{attribute addProperty BoxType "AX8206-0100-0101-0101"}
{attribute addProperty Id "DeviceDevice_F82A60211620Device_SafetyDevice_Safety_AF71BE9D160200Ch_ACh_A_359CD49A176220Ch_BCh_B_71B491C3176220WcStateAT %I*WcState_DC9C971540.50InfoDataAT %I*InfoData_17277C5A208260"}
{attribute addProperty CRC "932077249"}
{attribute addProperty SizeInBites "740"}
{attribute addProperty SizeInBytes "92.5"}
TYPE AX8206_36A80AF0 :
STRUCT
	{attribute addProperty Name "Device"}
	Device : Device_F82A6021;
	{attribute addProperty Name "Device_Safety"}
	Device_Safety : Device_Safety_AF71BE9D;
	{attribute addProperty Name "Ch_A"}
	Ch_A : Ch_A_359CD49A;
	{attribute addProperty Name "Ch_B"}
	Ch_B : Ch_B_71B491C3;
	{attribute addProperty Name "WcState"}
	WcState : WcState_DC9C9715;
	{attribute addProperty Name "InfoData"}
	InfoData : InfoData_17277C5A;
END_STRUCT
END_TYPE

(* stored: Version 1.2.0.0, ProductVersion 3.1.4024.9
   DUT AX8206_36A80AF0: Id {6e711265-d81c-4f7f-8bbc-49a74ca2f92f} *)
